LIN {X 0,Y 104.143,Z 808.734,A -85,B 0,C 180,E1 -870.899,E2 -870.899} C_VEL
LIN {X 0,Y 122.132,Z 801.22,A -85,B 0,C 180,E1 -878.965,E2 -878.965} C_VEL
LIN {X 0,Y 140.156,Z 792.678,A -85,B 0,C 180,E1 -884.394,E2 -884.394} C_VEL
LIN {X 0,Y 160.11,Z 781.742,A -85,B 0,C 180,E1 -888.665,E2 -888.665} C_VEL
LIN {X 0,Y 171.755,Z 774.595,A -85,B 0,C 180,E1 -890.616,E2 -890.616} C_VEL
LIN {X 0,Y 152.753,Z 784.632,A -85,B 0,C 180,E1 -894.259,E2 -894.259} C_VEL
LIN {X 0,Y 135.02,Z 792.507,A -85,B 0,C 180,E1 -898.779,E2 -898.779} C_VEL
LIN {X 0,Y 117.439,Z 799.027,A -85,B 0,C 180,E1 -904.996,E2 -904.996} C_VEL
LIN {X 0,Y 101.679,Z 803.804,A -85,B 0,C 180,E1 -913.193,E2 -913.193} C_VEL
LIN {X 0,Y 87.971,Z 806.999,A -85,B 0,C 180,E1 -924.581,E2 -924.581} C_VEL
LIN {X 0,Y 78.467,Z 808.347,A -85,B 0,C 180,E1 -938.975,E2 -938.975} C_VEL
LIN {X 0,Y 74.117,Z 808.088,A -85,B 0,C 180,E1 -954.534,E2 -954.534} C_VEL
LIN {X 0,Y 73.454,Z 806.99,A -85,B 0,C 180,E1 -966.741,E2 -966.741} C_VEL
LIN {X 0,Y 75.157,Z 804.666,A -85,B 0,C 180,E1 -980.806,E2 -980.806} C_VEL
LIN {X 0,Y 80.594,Z 800.783,A -85,B 0,C 180,E1 -994.974,E2 -994.974} C_VEL
LIN {X 0,Y 90.018,Z 795.001,A -85,B 0,C 180,E1 -1007.444,E2 -1007.444} C_VEL
LIN {X 0,Y 102.367,Z 787.467,A -85,B 0,C 180,E1 -1017.32,E2 -1017.32} C_VEL
LIN {X 0,Y 116.776,Z 778.007,A -85,B 0,C 180,E1 -1024.999,E2 -1024.999} C_VEL
LIN {X 0,Y 130.979,Z 767.68,A -85,B 0,C 180,E1 -1030.45,E2 -1030.45} C_VEL
LIN {X 0,Y 146.002,Z 755.346,A -85,B 0,C 180,E1 -1034.853,E2 -1034.853} C_VEL
LIN {X 0,Y 160.738,Z 741.468,A -85,B 0,C 180,E1 -1038.277,E2 -1038.277} C_VEL
LIN {X 0,Y 174.24,Z 726.949,A -85,B 0,C 180,E1 -1040.864,E2 -1040.864} C_VEL
LIN {X 0,Y 188.105,Z 709.776,A -85,B 0,C 180,E1 -1043.122,E2 -1043.122} C_VEL
LIN {X 0,Y 200.213,Z 692.322,A -85,B 0,C 180,E1 -1044.827,E2 -1044.827} C_VEL
LIN {X 0,Y 211.148,Z 673.87,A -85,B 0,C 180,E1 -1046.201,E2 -1046.201} C_VEL
LIN {X 0,Y 220.923,Z 654.057,A -85,B 0,C 180,E1 -1047.325,E2 -1047.325} C_VEL
LIN {X 0,Y 228.851,Z 634.412,A -85,B 0,C 180,E1 -1048.181,E2 -1048.181} C_VEL
LIN {X 0,Y 235.773,Z 612.825,A -85,B 0,C 180,E1 -1048.89,E2 -1048.89} C_VEL
LIN {X 0,Y 241.073,Z 590.503,A -85,B 0,C 180,E1 -1049.423,E2 -1049.423} C_VEL
LIN {X 0,Y 244.74,Z 567.255,A -85,B 0,C 180,E1 -1049.82,E2 -1049.82} C_VEL
LIN {X 0,Y 253.675,Z 495.963,A -85,B 0,C 180,E1 -1050.938,E2 -1050.938} C_VEL
LIN {X 0,Y 252.031,Z 491.853,A -85,B 0,C 180,E1 -1054.224,E2 -1054.224} C_VEL
LIN {X 0,Y 251.072,Z 489.341,A -85,B 0,C 180,E1 -1056.907,E2 -1056.907} C_VEL
LIN {X 0,Y 250.238,Z 486.677,A -85,B 0,C 180,E1 -1061.602,E2 -1061.602} C_VEL
LIN {X 0,Y 250.389,Z 486.91,A -85,B 0,C 180,E1 -1066.61,E2 -1066.61} C_VEL
LIN {X 0,Y 251.764,Z 490.567,A -85,B 0,C 180,E1 -1072.012,E2 -1072.012} C_VEL
LIN {X 0,Y 253.319,Z 494.346,A -85,B 0,C 180,E1 -1075.361,E2 -1075.361} C_VEL
LIN {X 0,Y 255.405,Z 499.347,A -85,B 0,C 180,E1 -1078.692,E2 -1078.692} C_VEL
LIN {X 0,Y 244.23,Z 589.375,A -85,B 0,C 180,E1 -1080.113,E2 -1080.113} C_VEL
LIN {X 0,Y 239.552,Z 611.763,A -85,B 0,C 180,E1 -1080.551,E2 -1080.551} C_VEL
LIN {X 0,Y 233.253,Z 633.14,A -85,B 0,C 180,E1 -1081.035,E2 -1081.035} C_VEL
LIN {X 0,Y 225.55,Z 653.583,A -85,B 0,C 180,E1 -1081.659,E2 -1081.659} C_VEL
LIN {X 0,Y 216.779,Z 672.714,A -85,B 0,C 180,E1 -1082.454,E2 -1082.454} C_VEL
LIN {X 0,Y 205.857,Z 692.548,A -85,B 0,C 180,E1 -1083.569,E2 -1083.569} C_VEL
LIN {X 0,Y 194.176,Z 710.425,A -85,B 0,C 180,E1 -1084.923,E2 -1084.923} C_VEL
LIN {X 0,Y 181.19,Z 727.592,A -85,B 0,C 180,E1 -1086.676,E2 -1086.676} C_VEL
LIN {X 0,Y 167.466,Z 743.395,A -85,B 0,C 180,E1 -1088.869,E2 -1088.869} C_VEL
LIN {X 0,Y 152.93,Z 758.082,A -85,B 0,C 180,E1 -1091.697,E2 -1091.697} C_VEL
LIN {X 0,Y 137.899,Z 771.353,A -85,B 0,C 180,E1 -1095.367,E2 -1095.367} C_VEL
LIN {X 0,Y 135.503,Z 773.384,A -85,B 0,C 180,E1 -1096.046,E2 -1096.046} C_VEL
LIN {X 0,Y 129.65,Z 777.607,A -85,B 0,C 180,E1 -1097.285,E2 -1097.285} C_VEL
LIN {X 0,Y 111.798,Z 787.807,A -85,B 0,C 180,E1 -1099.89,E2 -1099.89} C_VEL
LIN {X 0,Y 106.755,Z 790.847,A -85,B 0,C 180,E1 -1101.495,E2 -1101.495} C_VEL
LIN {X 0,Y 92.558,Z 799.689,A -85,B 0,C 180,E1 -1109.091,E2 -1109.091} C_VEL
LIN {X 0,Y 79.004,Z 807.674,A -85,B 0,C 180,E1 -1120.606,E2 -1120.606} C_VEL
LIN {X 0,Y 69.755,Z 813.442,A -85,B 0,C 180,E1 -1135.026,E2 -1135.026} C_VEL
LIN {X 0,Y 65.412,Z 817.223,A -85,B 0,C 180,E1 -1151.287,E2 -1151.287} C_VEL
LIN {X 0,Y 65.233,Z 819.3,A -85,B 0,C 180,E1 -1166.494,E2 -1166.494} C_VEL
LIN {X 0,Y 65.258,Z 819.678,A -85,B 0,C 180,E1 -1172.644,E2 -1172.644} C_VEL
LIN {X 0,Y 65.109,Z 819.693,A -85,B 0,C 180,E1 -1186.974,E2 -1186.974} C_VEL
LIN {X 0,Y 69.695,Z 818.157,A -85,B 0,C 180,E1 -1205.131,E2 -1205.131} C_VEL
LIN {X 0,Y 81.375,Z 814.648,A -85,B 0,C 180,E1 -1221.859,E2 -1221.859} C_VEL
LIN {X 0,Y 97.265,Z 809.482,A -85,B 0,C 180,E1 -1233.436,E2 -1233.436} C_VEL
LIN {X 0,Y 115.953,Z 802.46,A -85,B 0,C 180,E1 -1241.551,E2 -1241.551} C_VEL
LIN {X 0,Y 135.42,Z 793.877,A -85,B 0,C 180,E1 -1247.078,E2 -1247.078} C_VEL
LIN {X 0,Y 153.729,Z 784.586,A -85,B 0,C 180,E1 -1250.765,E2 -1250.765} C_VEL
LIN {X 0,Y 134.507,Z 792.925,A -85,B 0,C 180,E1 -1254.972,E2 -1254.972} C_VEL
LIN {X 0,Y 116,Z 799.521,A -85,B 0,C 180,E1 -1260.625,E2 -1260.625} C_VEL
LIN {X 0,Y 99.022,Z 804.373,A -85,B 0,C 180,E1 -1268.259,E2 -1268.259} C_VEL
LIN {X 0,Y 83.328,Z 807.683,A -85,B 0,C 180,E1 -1279.625,E2 -1279.625} C_VEL
LIN {X 0,Y 72.394,Z 809.064,A -85,B 0,C 180,E1 -1294.022,E2 -1294.022} C_VEL
LIN {X 0,Y 66.571,Z 808.89,A -85,B 0,C 180,E1 -1311.341,E2 -1311.341} C_VEL
LIN {X 0,Y 65.455,Z 807.85,A -85,B 0,C 180,E1 -1324.668,E2 -1324.668} C_VEL
LIN {X 0,Y 66.818,Z 805.812,A -85,B 0,C 180,E1 -1339.647,E2 -1339.647} C_VEL
LIN {X 0,Y 72.323,Z 802.011,A -85,B 0,C 180,E1 -1355.581,E2 -1355.581} C_VEL
LIN {X 0,Y 82.191,Z 796.462,A -85,B 0,C 180,E1 -1369.167,E2 -1369.167} C_VEL
LIN {X 0,Y 95.164,Z 789.17,A -85,B 0,C 180,E1 -1379.584,E2 -1379.584} C_VEL
LIN {X 0,Y 109.411,Z 780.502,A -85,B 0,C 180,E1 -1387.088,E2 -1387.088} C_VEL
LIN {X 0,Y 124.907,Z 769.869,A -85,B 0,C 180,E1 -1392.868,E2 -1392.868} C_VEL
LIN {X 0,Y 139.495,Z 758.476,A -85,B 0,C 180,E1 -1396.972,E2 -1396.972} C_VEL
LIN {X 0,Y 154.572,Z 745.1,A -85,B 0,C 180,E1 -1400.325,E2 -1400.325} C_VEL
LIN {X 0,Y 169.098,Z 730.32,A -85,B 0,C 180,E1 -1402.955,E2 -1402.955} C_VEL
LIN {X 0,Y 182.934,Z 714.072,A -85,B 0,C 180,E1 -1405.063,E2 -1405.063} C_VEL
LIN {X 0,Y 195.989,Z 696.094,A -85,B 0,C 180,E1 -1406.783,E2 -1406.783} C_VEL
LIN {X 0,Y 207.265,Z 677.783,A -85,B 0,C 180,E1 -1408.1,E2 -1408.1} C_VEL
LIN {X 0,Y 217.141,Z 658.766,A -85,B 0,C 180,E1 -1409.152,E2 -1409.152} C_VEL
LIN {X 0,Y 225.691,Z 638.857,A -85,B 0,C 180,E1 -1410.003,E2 -1410.003} C_VEL
LIN {X 0,Y 232.885,Z 617.918,A -85,B 0,C 180,E1 -1410.68,E2 -1410.68} C_VEL
LIN {X 0,Y 238.666,Z 595.537,A -85,B 0,C 180,E1 -1411.209,E2 -1411.209} C_VEL
LIN {X 0,Y 242.581,Z 572.938,A -85,B 0,C 180,E1 -1411.588,E2 -1411.588} C_VEL
LIN {X 0,Y 251.64,Z 501.944,A -85,B 0,C 180,E1 -1412.614,E2 -1412.614} C_VEL
LIN {X 0,Y 250.183,Z 497.757,A -85,B 0,C 180,E1 -1416.309,E2 -1416.309} C_VEL
LIN {X 0,Y 249.156,Z 494.592,A -85,B 0,C 180,E1 -1421.761,E2 -1421.761} C_VEL
LIN {X 0,Y 249.29,Z 494.743,A -85,B 0,C 180,E1 -1426.314,E2 -1426.314} C_VEL
LIN {X 0,Y 250.561,Z 498.396,A -85,B 0,C 180,E1 -1431.724,E2 -1431.724} C_VEL
LIN {X 0,Y 252.009,Z 502.096,A -85,B 0,C 180,E1 -1434.994,E2 -1434.994} C_VEL
LIN {X 0,Y 253.156,Z 505.112,A -85,B 0,C 180,E1 -1437.008,E2 -1437.008} C_VEL
LIN {X 0,Y 242.532,Z 589.057,A -85,B 0,C 180,E1 -1438.268,E2 -1438.268} C_VEL
LIN {X 0,Y 237.798,Z 611.401,A -85,B 0,C 180,E1 -1438.675,E2 -1438.675} C_VEL
LIN {X 0,Y 231.482,Z 632.612,A -85,B 0,C 180,E1 -1439.109,E2 -1439.109} C_VEL
LIN {X 0,Y 223.459,Z 653.622,A -85,B 0,C 180,E1 -1439.688,E2 -1439.688} C_VEL
LIN {X 0,Y 214.462,Z 672.874,A -85,B 0,C 180,E1 -1440.42,E2 -1440.42} C_VEL
LIN {X 0,Y 203.696,Z 692.129,A -85,B 0,C 180,E1 -1441.409,E2 -1441.409} C_VEL
LIN {X 0,Y 191.372,Z 710.666,A -85,B 0,C 180,E1 -1442.698,E2 -1442.698} C_VEL
LIN {X 0,Y 178.459,Z 727.376,A -85,B 0,C 180,E1 -1444.276,E2 -1444.276} C_VEL
LIN {X 0,Y 163.98,Z 743.636,A -85,B 0,C 180,E1 -1446.38,E2 -1446.38} C_VEL
LIN {X 0,Y 149.77,Z 757.629,A -85,B 0,C 180,E1 -1448.9,E2 -1448.9} C_VEL
LIN {X 0,Y 134.094,Z 771.039,A -85,B 0,C 180,E1 -1452.392,E2 -1452.392} C_VEL
LIN {X 0,Y 118.178,Z 783.031,A -85,B 0,C 180,E1 -1457.069,E2 -1457.069} C_VEL
LIN {X 0,Y 106.755,Z 790.847,A -85,B 0,C 180,E1 -1461.495,E2 -1461.495} C_VEL
LIN {X 0,Y 100.847,Z 794.254,A -85,B 0,C 180,E1 -1463.542,E2 -1463.542} C_VEL
LIN {X 0,Y 82.913,Z 801.991,A -85,B 0,C 180,E1 -1468.844,E2 -1468.844} C_VEL
LIN {X 0,Y 78.142,Z 804.207,A -85,B 0,C 180,E1 -1471.745,E2 -1471.745} C_VEL
LIN {X 0,Y 65.898,Z 810.78,A -85,B 0,C 180,E1 -1485.75,E2 -1485.75} C_VEL
LIN {X 0,Y 58.644,Z 815.414,A -85,B 0,C 180,E1 -1503.698,E2 -1503.698} C_VEL
LIN {X 0,Y 56.999,Z 817.933,A -85,B 0,C 180,E1 -1520.927,E2 -1520.927} C_VEL
LIN {X 0,Y 57.431,Z 818.734,A -85,B 0,C 180,E1 -1530.01,E2 -1530.01} C_VEL
LIN {X 0,Y 56.909,Z 819.017,A -85,B 0,C 180,E1 -1542.182,E2 -1542.182} C_VEL
LIN {X 0,Y 60.002,Z 818.27,A -85,B 0,C 180,E1 -1561.79,E2 -1561.79} C_VEL
LIN {X 0,Y 70.182,Z 815.754,A -85,B 0,C 180,E1 -1580.305,E2 -1580.305} C_VEL
LIN {X 0,Y 86.202,Z 811.392,A -85,B 0,C 180,E1 -1593.842,E2 -1593.842} C_VEL
LIN {X 0,Y 104.784,Z 805.448,A -85,B 0,C 180,E1 -1602.611,E2 -1602.611} C_VEL
LIN {X 0,Y 125.426,Z 797.473,A -85,B 0,C 180,E1 -1608.693,E2 -1608.693} C_VEL
LIN {X 0,Y 135.688,Z 792.959,A -85,B 0,C 180,E1 -1610.926,E2 -1610.926} C_VEL
LIN {X 0,Y 116.296,Z 799.734,A -85,B 0,C 180,E1 -1615.859,E2 -1615.859} C_VEL
LIN {X 0,Y 97.137,Z 804.93,A -85,B 0,C 180,E1 -1623.092,E2 -1623.092} C_VEL
LIN {X 0,Y 80.2,Z 808.233,A -85,B 0,C 180,E1 -1633.454,E2 -1633.454} C_VEL
LIN {X 0,Y 66.947,Z 809.793,A -85,B 0,C 180,E1 -1648.198,E2 -1648.198} C_VEL
LIN {X 0,Y 59.226,Z 809.686,A -85,B 0,C 180,E1 -1667.511,E2 -1667.511} C_VEL
LIN {X 0,Y 57.494,Z 808.613,A -85,B 0,C 180,E1 -1683.107,E2 -1683.107} C_VEL
LIN {X 0,Y 58.648,Z 806.731,A -85,B 0,C 180,E1 -1699.181,E2 -1699.181} C_VEL
LIN {X 0,Y 64.437,Z 803.026,A -85,B 0,C 180,E1 -1717.121,E2 -1717.121} C_VEL
LIN {X 0,Y 75.068,Z 797.589,A -85,B 0,C 180,E1 -1731.888,E2 -1731.888} C_VEL
LIN {X 0,Y 88.132,Z 790.854,A -85,B 0,C 180,E1 -1742.214,E2 -1742.214} C_VEL
LIN {X 0,Y 103.839,Z 781.874,A -85,B 0,C 180,E1 -1750.168,E2 -1750.168} C_VEL
LIN {X 0,Y 119.94,Z 771.354,A -85,B 0,C 180,E1 -1755.793,E2 -1755.793} C_VEL
LIN {X 0,Y 135.887,Z 759.416,A -85,B 0,C 180,E1 -1759.92,E2 -1759.92} C_VEL
LIN {X 0,Y 152.295,Z 745.229,A -85,B 0,C 180,E1 -1763.215,E2 -1763.215} C_VEL
LIN {X 0,Y 167.162,Z 730.345,A -85,B 0,C 180,E1 -1765.625,E2 -1765.625} C_VEL
LIN {X 0,Y 180.799,Z 714.591,A -85,B 0,C 180,E1 -1767.489,E2 -1767.489} C_VEL
LIN {X 0,Y 194.077,Z 696.59,A -85,B 0,C 180,E1 -1769.062,E2 -1769.062} C_VEL
LIN {X 0,Y 205.045,Z 679.076,A -85,B 0,C 180,E1 -1770.217,E2 -1770.217} C_VEL
LIN {X 0,Y 215.575,Z 659.156,A -85,B 0,C 180,E1 -1771.228,E2 -1771.228} C_VEL
LIN {X 0,Y 224.451,Z 638.655,A -85,B 0,C 180,E1 -1772.023,E2 -1772.023} C_VEL
LIN {X 0,Y 231.661,Z 617.752,A -85,B 0,C 180,E1 -1772.636,E2 -1772.636} C_VEL
LIN {X 0,Y 237.414,Z 595.626,A -85,B 0,C 180,E1 -1773.112,E2 -1773.112} C_VEL
LIN {X 0,Y 241.387,Z 572.834,A -85,B 0,C 180,E1 -1773.463,E2 -1773.463} C_VEL
LIN {X 0,Y 249.772,Z 507.924,A -85,B 0,C 180,E1 -1774.355,E2 -1774.355} C_VEL
LIN {X 0,Y 248.72,Z 504.93,A -85,B 0,C 180,E1 -1777.551,E2 -1777.551} C_VEL
LIN {X 0,Y 248.075,Z 502.508,A -85,B 0,C 180,E1 -1781.922,E2 -1781.922} C_VEL
LIN {X 0,Y 248.211,Z 502.699,A -85,B 0,C 180,E1 -1786.253,E2 -1786.253} C_VEL
LIN {X 0,Y 249.338,Z 506.137,A -85,B 0,C 180,E1 -1791.353,E2 -1791.353} C_VEL
LIN {X 0,Y 250.712,Z 509.844,A -85,B 0,C 180,E1 -1794.624,E2 -1794.624} C_VEL
LIN {X 0,Y 251.029,Z 510.928,A -85,B 0,C 180,E1 -1795.3,E2 -1795.3} C_VEL
LIN {X 0,Y 240.999,Z 588.8,A -85,B 0,C 180,E1 -1796.404,E2 -1796.404} C_VEL
LIN {X 0,Y 236.202,Z 611.184,A -85,B 0,C 180,E1 -1796.778,E2 -1796.778} C_VEL
LIN {X 0,Y 229.988,Z 631.881,A -85,B 0,C 180,E1 -1797.154,E2 -1797.154} C_VEL
LIN {X 0,Y 221.727,Z 653.345,A -85,B 0,C 180,E1 -1797.676,E2 -1797.676} C_VEL
LIN {X 0,Y 212.547,Z 672.743,A -85,B 0,C 180,E1 -1798.333,E2 -1798.333} C_VEL
LIN {X 0,Y 201.572,Z 692.111,A -85,B 0,C 180,E1 -1799.227,E2 -1799.227} C_VEL
LIN {X 0,Y 189.523,Z 709.964,A -85,B 0,C 180,E1 -1800.342,E2 -1800.342} C_VEL
LIN {X 0,Y 176.05,Z 727.118,A -85,B 0,C 180,E1 -1801.806,E2 -1801.806} C_VEL
LIN {X 0,Y 160.816,Z 743.815,A -85,B 0,C 180,E1 -1803.788,E2 -1803.788} C_VEL
LIN {X 0,Y 145.819,Z 758.096,A -85,B 0,C 180,E1 -1806.195,E2 -1806.195} C_VEL
LIN {X 0,Y 129.738,Z 771.417,A -85,B 0,C 180,E1 -1809.469,E2 -1809.469} C_VEL
LIN {X 0,Y 113.298,Z 783.246,A -85,B 0,C 180,E1 -1813.917,E2 -1813.917} C_VEL
LIN {X 0,Y 96.915,Z 793.635,A -85,B 0,C 180,E1 -1820.164,E2 -1820.164} C_VEL
LIN {X 0,Y 82.061,Z 802.099,A -85,B 0,C 180,E1 -1828.701,E2 -1828.701} C_VEL
LIN {X 0,Y 78.142,Z 804.207,A -85,B 0,C 180,E1 -1831.745,E2 -1831.745} C_VEL
LIN {X 0,Y 72.73,Z 806.663,A -85,B 0,C 180,E1 -1835.543,E2 -1835.543} C_VEL
LIN {X 0,Y 56.486,Z 811.92,A -85,B 0,C 180,E1 -1847.759,E2 -1847.759} C_VEL
LIN {X 0,Y 53.447,Z 813.157,A -85,B 0,C 180,E1 -1853.147,E2 -1853.147} C_VEL
LIN {X 0,Y 49.13,Z 816.572,A -85,B 0,C 180,E1 -1874.672,E2 -1874.672} C_VEL
LIN {X 0,Y 49.461,Z 817.926,A -85,B 0,C 180,E1 -1890.012,E2 -1890.012} C_VEL
LIN {X 0,Y 49.106,Z 818.223,A -85,B 0,C 180,E1 -1906.575,E2 -1906.575} C_VEL
LIN {X 0,Y 54.272,Z 817.38,A -85,B 0,C 180,E1 -1929.294,E2 -1929.294} C_VEL
LIN {X 0,Y 67.223,Z 814.724,A -85,B 0,C 180,E1 -1947.989,E2 -1947.989} C_VEL
LIN {X 0,Y 85.895,Z 810.104,A -85,B 0,C 180,E1 -1960.56,E2 -1960.56} C_VEL
LIN {X 0,Y 106.256,Z 803.898,A -85,B 0,C 180,E1 -1968.157,E2 -1968.157} C_VEL
LIN {X 0,Y 117.584,Z 799.86,A -85,B 0,C 180,E1 -1971.108,E2 -1971.108} C_VEL
LIN {X 0,Y 97.905,Z 805.054,A -85,B 0,C 180,E1 -1977.068,E2 -1977.068} C_VEL
LIN {X 0,Y 79.432,Z 808.596,A -85,B 0,C 180,E1 -1985.992,E2 -1985.992} C_VEL
LIN {X 0,Y 63.702,Z 810.45,A -85,B 0,C 180,E1 -1999.627,E2 -1999.627} C_VEL
LIN {X 0,Y 53.494,Z 810.653,A -85,B 0,C 180,E1 -2018.26,E2 -2018.26} C_VEL
LIN {X 0,Y 49.709,Z 809.574,A -85,B 0,C 180,E1 -2038.454,E2 -2038.454} C_VEL
LIN {X 0,Y 50.008,Z 808.033,A -85,B 0,C 180,E1 -2054.922,E2 -2054.922} C_VEL
LIN {X 0,Y 54.884,Z 804.926,A -85,B 0,C 180,E1 -2075.215,E2 -2075.215} C_VEL
LIN {X 0,Y 65.534,Z 799.934,A -85,B 0,C 180,E1 -2092.412,E2 -2092.412} C_VEL
LIN {X 0,Y 78.982,Z 793.557,A -85,B 0,C 180,E1 -2103.84,E2 -2103.84} C_VEL
LIN {X 0,Y 95.185,Z 785.084,A -85,B 0,C 180,E1 -2112.234,E2 -2112.234} C_VEL
LIN {X 0,Y 111.731,Z 775.173,A -85,B 0,C 180,E1 -2117.957,E2 -2117.957} C_VEL
LIN {X 0,Y 128.049,Z 763.908,A -85,B 0,C 180,E1 -2122.051,E2 -2122.051} C_VEL
LIN {X 0,Y 144.775,Z 750.411,A -85,B 0,C 180,E1 -2125.262,E2 -2125.262} C_VEL
LIN {X 0,Y 159.882,Z 736.249,A -85,B 0,C 180,E1 -2127.584,E2 -2127.584} C_VEL
LIN {X 0,Y 174.676,Z 720.19,A -85,B 0,C 180,E1 -2129.475,E2 -2129.475} C_VEL
LIN {X 0,Y 187.948,Z 703.408,A -85,B 0,C 180,E1 -2130.931,E2 -2130.931} C_VEL
LIN {X 0,Y 199.732,Z 686.046,A -85,B 0,C 180,E1 -2132.067,E2 -2132.067} C_VEL
LIN {X 0,Y 210.869,Z 666.438,A -85,B 0,C 180,E1 -2133.045,E2 -2133.045} C_VEL
LIN {X 0,Y 220.076,Z 646.812,A -85,B 0,C 180,E1 -2133.796,E2 -2133.796} C_VEL
LIN {X 0,Y 228.074,Z 625.701,A -85,B 0,C 180,E1 -2134.414,E2 -2134.414} C_VEL
LIN {X 0,Y 234.486,Z 603.658,A -85,B 0,C 180,E1 -2134.894,E2 -2134.894} C_VEL
LIN {X 0,Y 238.996,Z 581.99,A -85,B 0,C 180,E1 -2135.236,E2 -2135.236} C_VEL
LIN {X 0,Y 248.03,Z 514.263,A -85,B 0,C 180,E1 -2136.109,E2 -2136.109} C_VEL
LIN {X 0,Y 247.437,Z 512.377,A -85,B 0,C 180,E1 -2138.427,E2 -2138.427} C_VEL
LIN {X 0,Y 246.996,Z 510.424,A -85,B 0,C 180,E1 -2142.084,E2 -2142.084} C_VEL
LIN {X 0,Y 247.129,Z 510.67,A -85,B 0,C 180,E1 -2146.192,E2 -2146.192} C_VEL
LIN {X 0,Y 248.158,Z 513.986,A -85,B 0,C 180,E1 -2151.078,E2 -2151.078} C_VEL
LIN {X 0,Y 249.122,Z 516.737,A -85,B 0,C 180,E1 -2153.564,E2 -2153.564} C_VEL
LIN {X 0,Y 239.724,Z 588.387,A -85,B 0,C 180,E1 -2154.517,E2 -2154.517} C_VEL
LIN {X 0,Y 234.871,Z 610.785,A -85,B 0,C 180,E1 -2154.856,E2 -2154.856} C_VEL
LIN {X 0,Y 228.51,Z 631.759,A -85,B 0,C 180,E1 -2155.188,E2 -2155.188} C_VEL
LIN {X 0,Y 220.601,Z 652.178,A -85,B 0,C 180,E1 -2155.615,E2 -2155.615} C_VEL
LIN {X 0,Y 211.427,Z 671.535,A -85,B 0,C 180,E1 -2156.178,E2 -2156.178} C_VEL
LIN {X 0,Y 200.24,Z 691.138,A -85,B 0,C 180,E1 -2156.963,E2 -2156.963} C_VEL
LIN {X 0,Y 188.083,Z 709.015,A -85,B 0,C 180,E1 -2157.937,E2 -2157.937} C_VEL
LIN {X 0,Y 174.479,Z 726.191,A -85,B 0,C 180,E1 -2159.22,E2 -2159.22} C_VEL
LIN {X 0,Y 159.485,Z 742.475,A -85,B 0,C 180,E1 -2160.91,E2 -2160.91} C_VEL
LIN {X 0,Y 144.17,Z 756.899,A -85,B 0,C 180,E1 -2163.04,E2 -2163.04} C_VEL
LIN {X 0,Y 127.659,Z 770.277,A -85,B 0,C 180,E1 -2165.956,E2 -2165.956} C_VEL
LIN {X 0,Y 111.107,Z 781.889,A -85,B 0,C 180,E1 -2169.849,E2 -2169.849} C_VEL
LIN {X 0,Y 93.473,Z 792.658,A -85,B 0,C 180,E1 -2175.722,E2 -2175.722} C_VEL
LIN {X 0,Y 77.593,Z 801.198,A -85,B 0,C 180,E1 -2183.829,E2 -2183.829} C_VEL
LIN {X 0,Y 63.245,Z 808.255,A -85,B 0,C 180,E1 -2196.283,E2 -2196.283} C_VEL
LIN {X 0,Y 53.447,Z 813.157,A -85,B 0,C 180,E1 -2213.147,E2 -2213.147} C_VEL
LIN {X 0,Y 50.09,Z 814.727,A -85,B 0,C 180,E1 -2221.461,E2 -2221.461} C_VEL
LIN {X 0,Y 45.425,Z 816.195,A -85,B 0,C 180,E1 -2233.608,E2 -2233.608} C_VEL
LIN {X 0,Y 41.18,Z 817.243,A -85,B 0,C 180,E1 -2254.765,E2 -2254.765} C_VEL
LIN {X 0,Y 42.489,Z 817.355,A -85,B 0,C 180,E1 -2278.092,E2 -2278.092} C_VEL
LIN {X 0,Y 53.212,Z 815.896,A -85,B 0,C 180,E1 -2303.916,E2 -2303.916} C_VEL
LIN {X 0,Y 70.462,Z 812.73,A -85,B 0,C 180,E1 -2319.502,E2 -2319.502} C_VEL
LIN {X 0,Y 91.7,Z 807.563,A -85,B 0,C 180,E1 -2328.941,E2 -2328.941} C_VEL
LIN {X 0,Y 99.38,Z 805.282,A -85,B 0,C 180,E1 -2331.315,E2 -2331.315} C_VEL
LIN {X 0,Y 79.01,Z 809.117,A -85,B 0,C 180,E1 -2339.005,E2 -2339.005} C_VEL
LIN {X 0,Y 60.92,Z 811.168,A -85,B 0,C 180,E1 -2351.351,E2 -2351.351} C_VEL
LIN {X 0,Y 47.685,Z 811.434,A -85,B 0,C 180,E1 -2370.694,E2 -2370.694} C_VEL
LIN {X 0,Y 41.953,Z 810.338,A -85,B 0,C 180,E1 -2395.094,E2 -2395.094} C_VEL
LIN {X 0,Y 41.962,Z 808.782,A -85,B 0,C 180,E1 -2414.79,E2 -2414.79} C_VEL
LIN {X 0,Y 47.442,Z 805.681,A -85,B 0,C 180,E1 -2438.471,E2 -2438.471} C_VEL
LIN {X 0,Y 58.659,Z 800.966,A -85,B 0,C 180,E1 -2456.295,E2 -2456.295} C_VEL
LIN {X 0,Y 73.932,Z 794.337,A -85,B 0,C 180,E1 -2468.459,E2 -2468.459} C_VEL
LIN {X 0,Y 91.067,Z 785.888,A -85,B 0,C 180,E1 -2476.428,E2 -2476.428} C_VEL
LIN {X 0,Y 108.288,Z 776.004,A -85,B 0,C 180,E1 -2481.695,E2 -2481.695} C_VEL
LIN {X 0,Y 125.103,Z 764.758,A -85,B 0,C 180,E1 -2485.397,E2 -2485.397} C_VEL
LIN {X 0,Y 141.269,Z 752.079,A -85,B 0,C 180,E1 -2488.129,E2 -2488.129} C_VEL
LIN {X 0,Y 156.66,Z 738.115,A -85,B 0,C 180,E1 -2490.218,E2 -2490.218} C_VEL
LIN {X 0,Y 171.687,Z 722.292,A -85,B 0,C 180,E1 -2491.912,E2 -2491.912} C_VEL
LIN {X 0,Y 185.329,Z 705.541,A -85,B 0,C 180,E1 -2493.229,E2 -2493.229} C_VEL
LIN {X 0,Y 198.048,Z 687.136,A -85,B 0,C 180,E1 -2494.304,E2 -2494.304} C_VEL
LIN {X 0,Y 208.82,Z 668.535,A -85,B 0,C 180,E1 -2495.134,E2 -2495.134} C_VEL
LIN {X 0,Y 218.127,Z 649.297,A -85,B 0,C 180,E1 -2495.801,E2 -2495.801} C_VEL
LIN {X 0,Y 226.208,Z 628.766,A -85,B 0,C 180,E1 -2496.349,E2 -2496.349} C_VEL
LIN {X 0,Y 232.722,Z 607.561,A -85,B 0,C 180,E1 -2496.775,E2 -2496.775} C_VEL
LIN {X 0,Y 237.705,Z 585.023,A -85,B 0,C 180,E1 -2497.11,E2 -2497.11} C_VEL
LIN {X 0,Y 246.465,Z 520.713,A -85,B 0,C 180,E1 -2497.9,E2 -2497.9} C_VEL
LIN {X 0,Y 245.928,Z 518.356,A -85,B 0,C 180,E1 -2502.047,E2 -2502.047} C_VEL
LIN {X 0,Y 246.044,Z 518.645,A -85,B 0,C 180,E1 -2506.13,E2 -2506.13} C_VEL
LIN {X 0,Y 246.951,Z 521.707,A -85,B 0,C 180,E1 -2510.682,E2 -2510.682} C_VEL
LIN {X 0,Y 247.286,Z 523.017,A -85,B 0,C 180,E1 -2511.812,E2 -2511.812} C_VEL
LIN {X 0,Y 238.587,Z 588.228,A -85,B 0,C 180,E1 -2512.617,E2 -2512.617} C_VEL
LIN {X 0,Y 233.693,Z 610.594,A -85,B 0,C 180,E1 -2512.92,E2 -2512.92} C_VEL
LIN {X 0,Y 227.142,Z 631.952,A -85,B 0,C 180,E1 -2513.206,E2 -2513.206} C_VEL
LIN {X 0,Y 218.828,Z 653.039,A -85,B 0,C 180,E1 -2513.581,E2 -2513.581} C_VEL
LIN {X 0,Y 209.069,Z 673.092,A -85,B 0,C 180,E1 -2514.089,E2 -2514.089} C_VEL
LIN {X 0,Y 198.297,Z 691.613,A -85,B 0,C 180,E1 -2514.732,E2 -2514.732} C_VEL
LIN {X 0,Y 185.506,Z 710.083,A -85,B 0,C 180,E1 -2515.609,E2 -2515.609} C_VEL
LIN {X 0,Y 171.744,Z 726.987,A -85,B 0,C 180,E1 -2516.725,E2 -2516.725} C_VEL
LIN {X 0,Y 156.813,Z 742.782,A -85,B 0,C 180,E1 -2518.176,E2 -2518.176} C_VEL
LIN {X 0,Y 140.968,Z 757.274,A -85,B 0,C 180,E1 -2520.085,E2 -2520.085} C_VEL
LIN {X 0,Y 124.107,Z 770.571,A -85,B 0,C 180,E1 -2522.685,E2 -2522.685} C_VEL
LIN {X 0,Y 106.621,Z 782.341,A -85,B 0,C 180,E1 -2526.316,E2 -2526.316} C_VEL
LIN {X 0,Y 88.798,Z 792.66,A -85,B 0,C 180,E1 -2531.625,E2 -2531.625} C_VEL
LIN {X 0,Y 71.225,Z 801.432,A -85,B 0,C 180,E1 -2539.884,E2 -2539.884} C_VEL
LIN {X 0,Y 56.538,Z 808.003,A -85,B 0,C 180,E1 -2552.051,E2 -2552.051} C_VEL
LIN {X 0,Y 45.277,Z 813.013,A -85,B 0,C 180,E1 -2571.823,E2 -2571.823} C_VEL
LIN {X 0,Y 41.062,Z 816.155,A -85,B 0,C 180,E1 -2597.356,E2 -2597.356} C_VEL
LIN {X 0,Y 41.485,Z 817.111,A -85,B 0,C 180,E1 -2610.014,E2 -2610.014} C_VEL
LIN {X 0,Y 41.18,Z 817.243,A -85,B 0,C 180,E1 -2614.765,E2 -2614.765} C_VEL
LIN {X 0,Y 40.216,Z 817.382,A -85,B 0,C 180,E1 -2624.811,E2 -2624.811} C_VEL
LIN {X 0,Y 38.779,Z 816.936,A -85,B 0,C 180,E1 -2641.786,E2 -2641.786} C_VEL
LIN {X 0,Y 40.781,Z 816.243,A -85,B 0,C 180,E1 -2658.633,E2 -2658.633} C_VEL
LIN {X 0,Y 43.386,Z 815.889,A -85,B 0,C 180,E1 -2664.507,E2 -2664.507} C_VEL
LIN {X 0,Y 61.802,Z 813.279,A -85,B 0,C 180,E1 -2682.685,E2 -2682.685} C_VEL
LIN {X 0,Y 81.271,Z 809.434,A -85,B 0,C 180,E1 -2691.505,E2 -2691.505} C_VEL
LIN {X 0,Y 61.019,Z 811.709,A -85,B 0,C 180,E1 -2701.4,E2 -2701.4} C_VEL
LIN {X 0,Y 44.349,Z 812.245,A -85,B 0,C 180,E1 -2718.714,E2 -2718.714} C_VEL
LIN {X 0,Y 34.877,Z 811.312,A -85,B 0,C 180,E1 -2746.502,E2 -2746.502} C_VEL
LIN {X 0,Y 33.716,Z 809.761,A -85,B 0,C 180,E1 -2771.57,E2 -2771.57} C_VEL
LIN {X 0,Y 38.199,Z 807.21,A -85,B 0,C 180,E1 -2797.504,E2 -2797.504} C_VEL
LIN {X 0,Y 50.52,Z 802.571,A -85,B 0,C 180,E1 -2819.466,E2 -2819.466} C_VEL
LIN {X 0,Y 66.823,Z 796.215,A -85,B 0,C 180,E1 -2832.311,E2 -2832.311} C_VEL
LIN {X 0,Y 83.799,Z 788.576,A -85,B 0,C 180,E1 -2839.773,E2 -2839.773} C_VEL
LIN {X 0,Y 102.484,Z 778.516,A -85,B 0,C 180,E1 -2845.026,E2 -2845.026} C_VEL
LIN {X 0,Y 119.704,Z 767.539,A -85,B 0,C 180,E1 -2848.417,E2 -2848.417} C_VEL
LIN {X 0,Y 137.157,Z 754.513,A -85,B 0,C 180,E1 -2851.009,E2 -2851.009} C_VEL
LIN {X 0,Y 153.782,Z 739.958,A -85,B 0,C 180,E1 -2852.957,E2 -2852.957} C_VEL
LIN {X 0,Y 168.528,Z 724.939,A -85,B 0,C 180,E1 -2854.386,E2 -2854.386} C_VEL
LIN {X 0,Y 182.826,Z 707.851,A -85,B 0,C 180,E1 -2855.575,E2 -2855.575} C_VEL
LIN {X 0,Y 195.609,Z 689.798,A -85,B 0,C 180,E1 -2856.506,E2 -2856.506} C_VEL
LIN {X 0,Y 206.761,Z 671.147,A -85,B 0,C 180,E1 -2857.243,E2 -2857.243} C_VEL
LIN {X 0,Y 216.942,Z 650.624,A -85,B 0,C 180,E1 -2857.869,E2 -2857.869} C_VEL
LIN {X 0,Y 225.097,Z 630.318,A -85,B 0,C 180,E1 -2858.343,E2 -2858.343} C_VEL
LIN {X 0,Y 231.881,Z 608.631,A -85,B 0,C 180,E1 -2858.727,E2 -2858.727} C_VEL
LIN {X 0,Y 236.937,Z 586.058,A -85,B 0,C 180,E1 -2859.025,E2 -2859.025} C_VEL
LIN {X 0,Y 243.929,Z 535.998,A -85,B 0,C 180,E1 -2859.548,E2 -2859.548} C_VEL
LIN {X 0,Y 245.036,Z 527.613,A -85,B 0,C 180,E1 -2859.672,E2 -2859.672} C_VEL
LIN {X 0,Y 244.842,Z 526.266,A -85,B 0,C 180,E1 -2862.413,E2 -2862.413} C_VEL
LIN {X 0,Y 244.938,Z 526.461,A -85,B 0,C 180,E1 -2865.825,E2 -2865.825} C_VEL
LIN {X 0,Y 245.674,Z 529.292,A -85,B 0,C 180,E1 -2870.034,E2 -2870.034} C_VEL
LIN {X 0,Y 237.692,Z 588.018,A -85,B 0,C 180,E1 -2870.702,E2 -2870.702} C_VEL
LIN {X 0,Y 232.747,Z 610.372,A -85,B 0,C 180,E1 -2870.967,E2 -2870.967} C_VEL
LIN {X 0,Y 226.117,Z 631.792,A -85,B 0,C 180,E1 -2871.2,E2 -2871.2} C_VEL
LIN {X 0,Y 217.852,Z 652.588,A -85,B 0,C 180,E1 -2871.496,E2 -2871.496} C_VEL
LIN {X 0,Y 208.03,Z 672.628,A -85,B 0,C 180,E1 -2871.906,E2 -2871.906} C_VEL
LIN {X 0,Y 197.249,Z 691.027,A -85,B 0,C 180,E1 -2872.429,E2 -2872.429} C_VEL
LIN {X 0,Y 184.275,Z 709.606,A -85,B 0,C 180,E1 -2873.154,E2 -2873.154} C_VEL
LIN {X 0,Y 170.372,Z 726.522,A -85,B 0,C 180,E1 -2874.08,E2 -2874.08} C_VEL
LIN {X 0,Y 155.17,Z 742.405,A -85,B 0,C 180,E1 -2875.296,E2 -2875.296} C_VEL
LIN {X 0,Y 139.173,Z 756.809,A -85,B 0,C 180,E1 -2876.889,E2 -2876.889} C_VEL
LIN {X 0,Y 121.986,Z 770.098,A -85,B 0,C 180,E1 -2879.083,E2 -2879.083} C_VEL
LIN {X 0,Y 103.938,Z 781.909,A -85,B 0,C 180,E1 -2882.21,E2 -2882.21} C_VEL
LIN {X 0,Y 85.968,Z 791.924,A -85,B 0,C 180,E1 -2886.684,E2 -2886.684} C_VEL
LIN {X 0,Y 67.036,Z 800.87,A -85,B 0,C 180,E1 -2894.23,E2 -2894.23} C_VEL
LIN {X 0,Y 51.083,Z 807.392,A -85,B 0,C 180,E1 -2905.822,E2 -2905.822} C_VEL
LIN {X 0,Y 38.104,Z 812.401,A -85,B 0,C 180,E1 -2927.003,E2 -2927.003} C_VEL
LIN {X 0,Y 33.085,Z 815.493,A -85,B 0,C 180,E1 -2957.806,E2 -2957.806} C_VEL
LIN {X 0,Y 33.495,Z 816.288,A -85,B 0,C 180,E1 -2970.018,E2 -2970.018} C_VEL
LIN {X 0,Y 34.511,Z 816.63,A -85,B 0,C 180,E1 -2999.612,E2 -2999.612} C_VEL
LIN {X 0,Y 43.386,Z 815.889,A -85,B 0,C 180,E1 -3024.507,E2 -3024.507} C_VEL
LIN {X 0,Y 46.039,Z 815.491,A -85,B 0,C 180,E1 -3030.262,E2 -3030.262} C_VEL
LIN {X 0,Y 52.435,Z 813.875,A -85,B 0,C 180,E1 -3045.335,E2 -3045.335} C_VEL
LIN {X 0,Y 55.893,Z 813.349,A -85,B 0,C 180,E1 -3048.327,E2 -3048.327} C_VEL
LIN {X 0,Y 62.881,Z 812.234,A -85,B 0,C 180,E1 -3051.765,E2 -3051.765} C_VEL
LIN {X 0,Y 43.194,Z 813.07,A -85,B 0,C 180,E1 -3065.383,E2 -3065.383} C_VEL
LIN {X 0,Y 29.41,Z 812.347,A -85,B 0,C 180,E1 -3091.758,E2 -3091.758} C_VEL
LIN {X 0,Y 25.564,Z 810.845,A -85,B 0,C 180,E1 -3124.492,E2 -3124.492} C_VEL
LIN {X 0,Y 29.22,Z 808.539,A -85,B 0,C 180,E1 -3157.241,E2 -3157.241} C_VEL
LIN {X 0,Y 41.995,Z 804.357,A -85,B 0,C 180,E1 -3183.185,E2 -3183.185} C_VEL
LIN {X 0,Y 59.174,Z 798.393,A -85,B 0,C 180,E1 -3196.584,E2 -3196.584} C_VEL
LIN {X 0,Y 76.853,Z 791.02,A -85,B 0,C 180,E1 -3203.753,E2 -3203.753} C_VEL
LIN {X 0,Y 96.087,Z 781.404,A -85,B 0,C 180,E1 -3208.557,E2 -3208.557} C_VEL
LIN {X 0,Y 114.667,Z 770.273,A -85,B 0,C 180,E1 -3211.713,E2 -3211.713} C_VEL
LIN {X 0,Y 131.612,Z 758.323,A -85,B 0,C 180,E1 -3213.861,E2 -3213.861} C_VEL
LIN {X 0,Y 148.287,Z 744.452,A -85,B 0,C 180,E1 -3215.531,E2 -3215.531} C_VEL
LIN {X 0,Y 163.697,Z 729.447,A -85,B 0,C 180,E1 -3216.806,E2 -3216.806} C_VEL
LIN {X 0,Y 178.495,Z 712.605,A -85,B 0,C 180,E1 -3217.851,E2 -3217.851} C_VEL
LIN {X 0,Y 191.604,Z 695.079,A -85,B 0,C 180,E1 -3218.656,E2 -3218.656} C_VEL
LIN {X 0,Y 203.08,Z 677.035,A -85,B 0,C 180,E1 -3219.292,E2 -3219.292} C_VEL
LIN {X 0,Y 213.551,Z 657.167,A -85,B 0,C 180,E1 -3219.833,E2 -3219.833} C_VEL
LIN {X 0,Y 222.012,Z 637.515,A -85,B 0,C 180,E1 -3220.254,E2 -3220.254} C_VEL
LIN {X 0,Y 229.5,Z 615.547,A -85,B 0,C 180,E1 -3220.613,E2 -3220.613} C_VEL
LIN {X 0,Y 235.079,Z 593.458,A -85,B 0,C 180,E1 -3220.885,E2 -3220.885} C_VEL
LIN {X 0,Y 238.934,Z 570.794,A -85,B 0,C 180,E1 -3221.104,E2 -3221.104} C_VEL
LIN {X 0,Y 243.795,Z 534.519,A -85,B 0,C 180,E1 -3221.47,E2 -3221.47} C_VEL
LIN {X 0,Y 243.774,Z 534.164,A -85,B 0,C 180,E1 -3224.784,E2 -3224.784} C_VEL
LIN {X 0,Y 243.985,Z 535.356,A -85,B 0,C 180,E1 -3227.233,E2 -3227.233} C_VEL
LIN {X 0,Y 244.127,Z 536.168,A -85,B 0,C 180,E1 -3228.242,E2 -3228.242} C_VEL
LIN {X 0,Y 236.97,Z 587.906,A -85,B 0,C 180,E1 -3228.777,E2 -3228.777} C_VEL
LIN {X 0,Y 231.964,Z 610.346,A -85,B 0,C 180,E1 -3229.004,E2 -3229.004} C_VEL
LIN {X 0,Y 225.208,Z 631.953,A -85,B 0,C 180,E1 -3229.182,E2 -3229.182} C_VEL
LIN {X 0,Y 217.217,Z 651.924,A -85,B 0,C 180,E1 -3229.392,E2 -3229.392} C_VEL
LIN {X 0,Y 207.1,Z 672.461,A -85,B 0,C 180,E1 -3229.712,E2 -3229.712} C_VEL
LIN {X 0,Y 195.857,Z 691.41,A -85,B 0,C 180,E1 -3230.133,E2 -3230.133} C_VEL
LIN {X 0,Y 182.868,Z 709.823,A -85,B 0,C 180,E1 -3230.696,E2 -3230.696} C_VEL
LIN {X 0,Y 168.851,Z 726.608,A -85,B 0,C 180,E1 -3231.426,E2 -3231.426} C_VEL
LIN {X 0,Y 153.312,Z 742.56,A -85,B 0,C 180,E1 -3232.404,E2 -3232.404} C_VEL
LIN {X 0,Y 136.792,Z 757.099,A -85,B 0,C 180,E1 -3233.71,E2 -3233.71} C_VEL
LIN {X 0,Y 119.341,Z 770.243,A -85,B 0,C 180,E1 -3235.49,E2 -3235.49} C_VEL
LIN {X 0,Y 101.033,Z 781.916,A -85,B 0,C 180,E1 -3238.036,E2 -3238.036} C_VEL
LIN {X 0,Y 83.011,Z 791.575,A -85,B 0,C 180,E1 -3241.645,E2 -3241.645} C_VEL
LIN {X 0,Y 63.582,Z 800.298,A -85,B 0,C 180,E1 -3247.895,E2 -3247.895} C_VEL
LIN {X 0,Y 45.463,Z 807.062,A -85,B 0,C 180,E1 -3259.014,E2 -3259.014} C_VEL
LIN {X 0,Y 31.324,Z 811.77,A -85,B 0,C 180,E1 -3280.028,E2 -3280.028} C_VEL
LIN {X 0,Y 25.138,Z 814.703,A -85,B 0,C 180,E1 -3316.218,E2 -3316.218} C_VEL
LIN {X 0,Y 25.47,Z 815.395,A -85,B 0,C 180,E1 -3330.024,E2 -3330.024} C_VEL
LIN {X 0,Y 28.094,Z 815.836,A -85,B 0,C 180,E1 -3369.865,E2 -3369.865} C_VEL
LIN {X 0,Y 42.933,Z 814.873,A -85,B 0,C 180,E1 -3398.715,E2 -3398.715} C_VEL
LIN {X 0,Y 55.893,Z 813.349,A -85,B 0,C 180,E1 -3408.327,E2 -3408.327} C_VEL
LIN {X 0,Y 54.326,Z 813.418,A -85,B 0,C 180,E1 -3408.985,E2 -3408.985} C_VEL
LIN {X 0,Y 46.593,Z 814.03,A -85,B 0,C 180,E1 -3407.813,E2 -3407.813} C_VEL
LIN {X 0,Y 29.657,Z 814.922,A -85,B 0,C 180,E1 -3397.354,E2 -3397.354} C_VEL
LIN {X 0,Y 23.239,Z 815.033,A -85,B 0,C 180,E1 -3385.909,E2 -3385.909} C_VEL
LIN {X 0,Y 17.287,Z 814.565,A -85,B 0,C 180,E1 -3333.351,E2 -3333.351} C_VEL
LIN {X 0,Y 17.144,Z 814.142,A -85,B 0,C 180,E1 -3319.959,E2 -3319.959} C_VEL
LIN {X 0,Y 24.524,Z 811.35,A -85,B 0,C 180,E1 -3271.157,E2 -3271.157} C_VEL
LIN {X 0,Y 41.59,Z 806.434,A -85,B 0,C 180,E1 -3249.802,E2 -3249.802} C_VEL
LIN {X 0,Y 60.988,Z 799.69,A -85,B 0,C 180,E1 -3240.929,E2 -3240.929} C_VEL
LIN {X 0,Y 81.155,Z 790.988,A -85,B 0,C 180,E1 -3236.205,E2 -3236.205} C_VEL
LIN {X 0,Y 99.608,Z 781.351,A -85,B 0,C 180,E1 -3233.532,E2 -3233.532} C_VEL
LIN {X 0,Y 118.222,Z 769.689,A -85,B 0,C 180,E1 -3231.66,E2 -3231.66} C_VEL
LIN {X 0,Y 135.887,Z 756.542,A -85,B 0,C 180,E1 -3230.362,E2 -3230.362} C_VEL
LIN {X 0,Y 152.563,Z 741.991,A -85,B 0,C 180,E1 -3229.413,E2 -3229.413} C_VEL
LIN {X 0,Y 168.22,Z 726.017,A -85,B 0,C 180,E1 -3228.71,E2 -3228.71} C_VEL
LIN {X 0,Y 182.324,Z 709.197,A -85,B 0,C 180,E1 -3228.187,E2 -3228.187} C_VEL
LIN {X 0,Y 195.38,Z 690.772,A -85,B 0,C 180,E1 -3227.789,E2 -3227.789} C_VEL
LIN {X 0,Y 206.596,Z 671.938,A -85,B 0,C 180,E1 -3227.498,E2 -3227.498} C_VEL
LIN {X 0,Y 216.763,Z 651.369,A -85,B 0,C 180,E1 -3227.282,E2 -3227.282} C_VEL
LIN {X 0,Y 225.101,Z 630.438,A -85,B 0,C 180,E1 -3227.141,E2 -3227.141} C_VEL
LIN {X 0,Y 231.71,Z 609.098,A -85,B 0,C 180,E1 -3227.021,E2 -3227.021} C_VEL
LIN {X 0,Y 236.683,Z 586.784,A -85,B 0,C 180,E1 -3226.833,E2 -3226.833} C_VEL
LIN {X 0,Y 242.822,Z 542.843,A -85,B 0,C 180,E1 -3226.385,E2 -3226.385} C_VEL
LIN {X 0,Y 242.693,Z 542.082,A -85,B 0,C 180,E1 -3224.578,E2 -3224.578} C_VEL
LIN {X 0,Y 242.636,Z 542.266,A -85,B 0,C 180,E1 -3223.259,E2 -3223.259} C_VEL
LIN {X 0,Y 236.253,Z 587.006,A -85,B 0,C 180,E1 -3222.891,E2 -3222.891} C_VEL
LIN {X 0,Y 231.159,Z 609.478,A -85,B 0,C 180,E1 -3222.678,E2 -3222.678} C_VEL
LIN {X 0,Y 224.44,Z 630.747,A -85,B 0,C 180,E1 -3222.419,E2 -3222.419} C_VEL
LIN {X 0,Y 216.426,Z 650.621,A -85,B 0,C 180,E1 -3222.107,E2 -3222.107} C_VEL
LIN {X 0,Y 206.397,Z 670.823,A -85,B 0,C 180,E1 -3221.701,E2 -3221.701} C_VEL
LIN {X 0,Y 195.353,Z 689.32,A -85,B 0,C 180,E1 -3221.227,E2 -3221.227} C_VEL
LIN {X 0,Y 182.287,Z 707.7,A -85,B 0,C 180,E1 -3220.625,E2 -3220.625} C_VEL
LIN {X 0,Y 168.217,Z 724.386,A -85,B 0,C 180,E1 -3219.894,E2 -3219.894} C_VEL
LIN {X 0,Y 153.146,Z 739.695,A -85,B 0,C 180,E1 -3218.993,E2 -3218.993} C_VEL
LIN {X 0,Y 137.085,Z 753.711,A -85,B 0,C 180,E1 -3217.852,E2 -3217.852} C_VEL
LIN {X 0,Y 120.046,Z 766.441,A -85,B 0,C 180,E1 -3216.361,E2 -3216.361} C_VEL
LIN {X 0,Y 102.052,Z 777.731,A -85,B 0,C 180,E1 -3214.324,E2 -3214.324} C_VEL
LIN {X 0,Y 83.161,Z 787.675,A -85,B 0,C 180,E1 -3211.349,E2 -3211.349} C_VEL
LIN {X 0,Y 63.423,Z 796.221,A -85,B 0,C 180,E1 -3206.521,E2 -3206.521} C_VEL
LIN {X 0,Y 44.394,Z 802.892,A -85,B 0,C 180,E1 -3197.987,E2 -3197.987} C_VEL
LIN {X 0,Y 27.685,Z 807.691,A -85,B 0,C 180,E1 -3179.951,E2 -3179.951} C_VEL
LIN {X 0,Y 18.151,Z 810.712,A -85,B 0,C 180,E1 -3140.454,E2 -3140.454} C_VEL
LIN {X 0,Y 19.703,Z 812.401,A -85,B 0,C 180,E1 -3095.66,E2 -3095.66} C_VEL
LIN {X 0,Y 33.152,Z 813.735,A -85,B 0,C 180,E1 -3061.714,E2 -3061.714} C_VEL
LIN {X 0,Y 44.363,Z 813.885,A -85,B 0,C 180,E1 -3052.055,E2 -3052.055} C_VEL
LIN {X 0,Y 24.482,Z 814.999,A -85,B 0,C 180,E1 -3029.101,E2 -3029.101} C_VEL
LIN {X 0,Y 23.239,Z 815.033,A -85,B 0,C 180,E1 -3025.909,E2 -3025.909} C_VEL
LIN {X 0,Y 19.46,Z 814.953,A -85,B 0,C 180,E1 -3016.405,E2 -3016.405} C_VEL
LIN {X 0,Y 13.69,Z 814.403,A -85,B 0,C 180,E1 -2999.645,E2 -2999.645} C_VEL
LIN {X 0,Y 9.504,Z 813.074,A -85,B 0,C 180,E1 -2943.482,E2 -2943.482} C_VEL
LIN {X 0,Y 23.315,Z 809.809,A -85,B 0,C 180,E1 -2889.632,E2 -2889.632} C_VEL
LIN {X 0,Y 42.012,Z 804.959,A -85,B 0,C 180,E1 -2877.885,E2 -2877.885} C_VEL
LIN {X 0,Y 62.456,Z 797.924,A -85,B 0,C 180,E1 -2872.919,E2 -2872.919} C_VEL
LIN {X 0,Y 82.139,Z 789.389,A -85,B 0,C 180,E1 -2870.35,E2 -2870.35} C_VEL
LIN {X 0,Y 102.028,Z 778.843,A -85,B 0,C 180,E1 -2868.702,E2 -2868.702} C_VEL
LIN {X 0,Y 119.734,Z 767.646,A -85,B 0,C 180,E1 -2867.669,E2 -2867.669} C_VEL
LIN {X 0,Y 137.547,Z 754.275,A -85,B 0,C 180,E1 -2866.903,E2 -2866.903} C_VEL
LIN {X 0,Y 153.809,Z 739.89,A -85,B 0,C 180,E1 -2866.354,E2 -2866.354} C_VEL
LIN {X 0,Y 169.543,Z 723.625,A -85,B 0,C 180,E1 -2865.94,E2 -2865.94} C_VEL
LIN {X 0,Y 183.707,Z 706.443,A -85,B 0,C 180,E1 -2865.634,E2 -2865.634} C_VEL
LIN {X 0,Y 196.281,Z 688.511,A -85,B 0,C 180,E1 -2865.421,E2 -2865.421} C_VEL
LIN {X 0,Y 207.8,Z 668.842,A -85,B 0,C 180,E1 -2865.257,E2 -2865.257} C_VEL
LIN {X 0,Y 217.484,Z 648.742,A -85,B 0,C 180,E1 -2865.155,E2 -2865.155} C_VEL
LIN {X 0,Y 225.542,Z 628.007,A -85,B 0,C 180,E1 -2865.098,E2 -2865.098} C_VEL
LIN {X 0,Y 232.11,Z 606.095,A -85,B 0,C 180,E1 -2865.028,E2 -2865.028} C_VEL
LIN {X 0,Y 236.763,Z 584.486,A -85,B 0,C 180,E1 -2864.877,E2 -2864.877} C_VEL
LIN {X 0,Y 236.915,Z 583.509,A -85,B 0,C 180,E1 -2864.859,E2 -2864.859} C_VEL
LIN {X 0,Y 232.28,Z 605.259,A -85,B 0,C 180,E1 -2864.702,E2 -2864.702} C_VEL
LIN {X 0,Y 225.721,Z 627.262,A -85,B 0,C 180,E1 -2864.503,E2 -2864.503} C_VEL
LIN {X 0,Y 217.616,Z 648.159,A -85,B 0,C 180,E1 -2864.261,E2 -2864.261} C_VEL
LIN {X 0,Y 208.047,Z 668.037,A -85,B 0,C 180,E1 -2863.971,E2 -2863.971} C_VEL
LIN {X 0,Y 196.441,Z 687.793,A -85,B 0,C 180,E1 -2863.613,E2 -2863.613} C_VEL
LIN {X 0,Y 183.808,Z 705.757,A -85,B 0,C 180,E1 -2863.2,E2 -2863.2} C_VEL
LIN {X 0,Y 169.654,Z 722.863,A -85,B 0,C 180,E1 -2862.684,E2 -2862.684} C_VEL
LIN {X 0,Y 154.478,Z 738.52,A -85,B 0,C 180,E1 -2862.06,E2 -2862.06} C_VEL
LIN {X 0,Y 138.284,Z 752.833,A -85,B 0,C 180,E1 -2861.281,E2 -2861.281} C_VEL
LIN {X 0,Y 121.069,Z 765.712,A -85,B 0,C 180,E1 -2860.285,E2 -2860.285} C_VEL
LIN {X 0,Y 102.84,Z 777.241,A -85,B 0,C 180,E1 -2858.947,E2 -2858.947} C_VEL
LIN {X 0,Y 82.594,Z 787.889,A -85,B 0,C 180,E1 -2856.911,E2 -2856.911} C_VEL
LIN {X 0,Y 63.399,Z 796.138,A -85,B 0,C 180,E1 -2853.997,E2 -2853.997} C_VEL
LIN {X 0,Y 43.315,Z 803.025,A -85,B 0,C 180,E1 -2848.631,E2 -2848.631} C_VEL
LIN {X 0,Y 23.768,Z 808.13,A -85,B 0,C 180,E1 -2835.619,E2 -2835.619} C_VEL
LIN {X 0,Y 10.503,Z 811.292,A -85,B 0,C 180,E1 -2789.943,E2 -2789.943} C_VEL
LIN {X 0,Y 12.852,Z 812.937,A -85,B 0,C 180,E1 -2720.869,E2 -2720.869} C_VEL
LIN {X 0,Y 25.115,Z 814.131,A -85,B 0,C 180,E1 -2692.547,E2 -2692.547} C_VEL
LIN {X 0,Y 9.442,Z 813.859,A -85,B 0,C 180,E1 -2635.131,E2 -2635.131} C_VEL
LIN {X 0,Y 9.334,Z 813.57,A -85,B 0,C 180,E1 -2610.064,E2 -2610.064} C_VEL
LIN {X 0,Y 9.504,Z 813.074,A -85,B 0,C 180,E1 -2583.482,E2 -2583.482} C_VEL
LIN {X 0,Y 12.534,Z 812.038,A -85,B 0,C 180,E1 -2549.117,E2 -2549.117} C_VEL
LIN {X 0,Y 21.194,Z 809.629,A -85,B 0,C 180,E1 -2519.188,E2 -2519.188} C_VEL
LIN {X 0,Y 31.088,Z 806.986,A -85,B 0,C 180,E1 -2508.816,E2 -2508.816} C_VEL
LIN {X 0,Y 35.891,Z 805.673,A -85,B 0,C 180,E1 -2507.438,E2 -2507.438} C_VEL
LIN {X 0,Y 57.75,Z 798.805,A -85,B 0,C 180,E1 -2505.782,E2 -2505.782} C_VEL
LIN {X 0,Y 77.659,Z 790.731,A -85,B 0,C 180,E1 -2504.9,E2 -2504.9} C_VEL
LIN {X 0,Y 97.615,Z 780.712,A -85,B 0,C 180,E1 -2504.304,E2 -2504.304} C_VEL
LIN {X 0,Y 115.51,Z 769.79,A -85,B 0,C 180,E1 -2503.887,E2 -2503.887} C_VEL
LIN {X 0,Y 97.134,Z 780.845,A -85,B 0,C 180,E1 -2503.173,E2 -2503.173} C_VEL
LIN {X 0,Y 77.692,Z 790.483,A -85,B 0,C 180,E1 -2502.212,E2 -2502.212} C_VEL
LIN {X 0,Y 57.9,Z 798.414,A -85,B 0,C 180,E1 -2500.855,E2 -2500.855} C_VEL
LIN {X 0,Y 36.537,Z 805.094,A -85,B 0,C 180,E1 -2498.454,E2 -2498.454} C_VEL
LIN {X 0,Y 16.79,Z 809.702,A -85,B 0,C 180,E1 -2493.205,E2 -2493.205} C_VEL
LIN {X 0,Y 1.774,Z 812.299,A -85,B 0,C 180,E1 -2429.661,E2 -2429.661} C_VEL
LIN {X 0,Y 4.153,Z 812.935,A -85,B 0,C 180,E1 -2334.616,E2 -2334.616} C_VEL
LIN {X 0,Y 1.236,Z 812.644,A -85,B 0,C 180,E1 -2250.486,E2 -2250.486} C_VEL
LIN {X 0,Y 18.238,Z 809.805,A -85,B 0,C 180,E1 -2150.485,E2 -2150.485} C_VEL
LIN {X 0,Y 35.891,Z 805.673,A -85,B 0,C 180,E1 -2147.438,E2 -2147.438} C_VEL
LIN {X 0,Y 38.398,Z 807.607,A -85,B 0,C 180,E1 -2147.191,E2 -2147.191} C_VEL
LIN {X 0,Y 38.398,Z 862.5,A -85,B 0,C 180,E1 -2147.191,E2 -2147.191} C_VEL
LIN {X 0,Y 38.398,Z 862.5,A -85,B 0,C 180,E1 -2147.191,E2 -2147.191}

QRS_NEXT_CUT()

QRS_NEXT()
QRS_HOME()

END
